TYPE ST_IdentityOUT2 :
STRUCT
	ID	:STRING;
	ReadQuality:STRING;
END_STRUCT
END_TYPE

(* stored: Version 1.1.0.1, ProductVersion 3.1.4024.13
   DUT ST_IdentityOUT2: Id {2cec02a6-7c68-49d4-9994-7fe61b18a982} *)
